PROGRAM P_Control_Mode
VAR
END_VAR

// ***********************************************************************************
//
// Müller-steinag Gruppe, Kandergrien Einigen, CH-3646 Bern
// ETH Zurich, Building HIF E26, Laura-Hezner-Weg 7, CH-8093 Zürich
// 
// ***********************************************************************************
// 
// PROJECT     :  A061 Digital Casting System 
// FUNCTION    :  Control mode 
// AUTHOR      :  Weiting Chen
// EMAIL       :  chenw@usi.ch
// Copyright   :  USI Mendrisio; ETH Zürich; Müller-steinag Gruppe (CH) 2023
//
// ***********************************************************************************

GVL.b_mode_manual := GVL_IO.ib_CC1_Button_Mode_Manual; 
GVL.b_mode_laptop := GVL_IO.ib_CC1_Button_Mode_Laptop;



IF GVL.b_mode_manual THEN 
	GVL.s_current_mode := 'Controller';
ELSIF GVL.b_mode_laptop  THEN
	GVL.s_current_mode := 'Laptop';
ELSIF NOT GVL.b_mode_manual AND NOT GVL.b_mode_laptop THEN
	GVL.s_current_mode := 'Robot';
	GVL.b_mode_robot := TRUE;
ELSE
	GVL.s_current_mode := 'None';
END_IF

END_PROGRAM

(* stored: Version 1.1.0.1, ProductVersion 3.1.4024.11
   POU P_Control_Mode: Id {ee662d16-9f8f-400c-b3c1-3f76b012b61b}, SpecialFunc None *)
